Fanuc KAREL source: ka00092.KL

PROGRAM KA00092
%STACKSIZE=65535
%PRIORITY=65535
%NOLOCKGROUP
VAR
SRC : JOINTPOS9
DST : JOINTPOS9
BEGIN
DST=SRC
END KA00092
